// Mitsubishi GX Works2 project: Task Reverse 5 count p103   PLC: FX3S
// Task Reverse after 5 count p103

PROGRAM MAIN
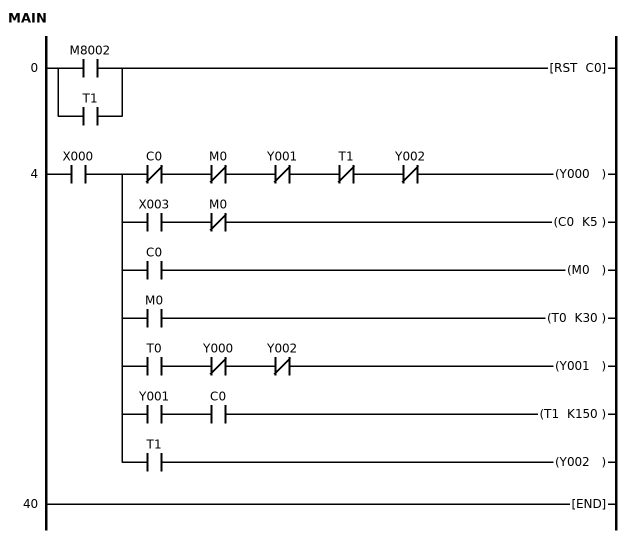
0     LD      M8002
      OR      T1
      RST     C0
4     LD      X000
      MPS
      ANI     C0
      ANI     M0
      ANI     Y001
      ANI     T1
      ANI     Y002
      OUT     Y000
      MRD
      AND     X003
      ANI     M0
      OUT     C0 K5
      MRD
      AND     C0
      OUT     M0
      MRD
      AND     M0
      OUT     T0 K30
      MRD
      AND     T0
      ANI     Y000
      ANI     Y002
      OUT     Y001
      MRD
      AND     Y001
      AND     C0
      OUT     T1 K150
      MPP
      AND     T1
      OUT     Y002
40    END
END_PROGRAM
